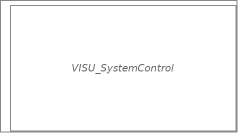
VISUALIZATION VISU_ServicesOverview  // 238x133
VAR_IN_OUT
    ref : Services;
    widget : ServicesWidget;
END_VAR
    Frame (10,5 226x126)
        shows VISU_SystemControl(status := widget.actualStatus, button_initialize := widget.button_initialize, button_operating := widget.button_operating, button_locking := widget.button_locking)
END_VISUALIZATION

(* stored: Version 1.1.0.1, ProductVersion 3.1.4019.2
   Visu VISU_ServicesOverview: Id {b180b128-3bab-4004-b389-e35d4ca5d594} *)
